REGION Network 112: SALIDAS - VELOCIDAD ANALOGICA >> RODILLOS
   // 25T229A_03 
   // Plantilla_Avance_E1S3_SinVariador_1Mesas.
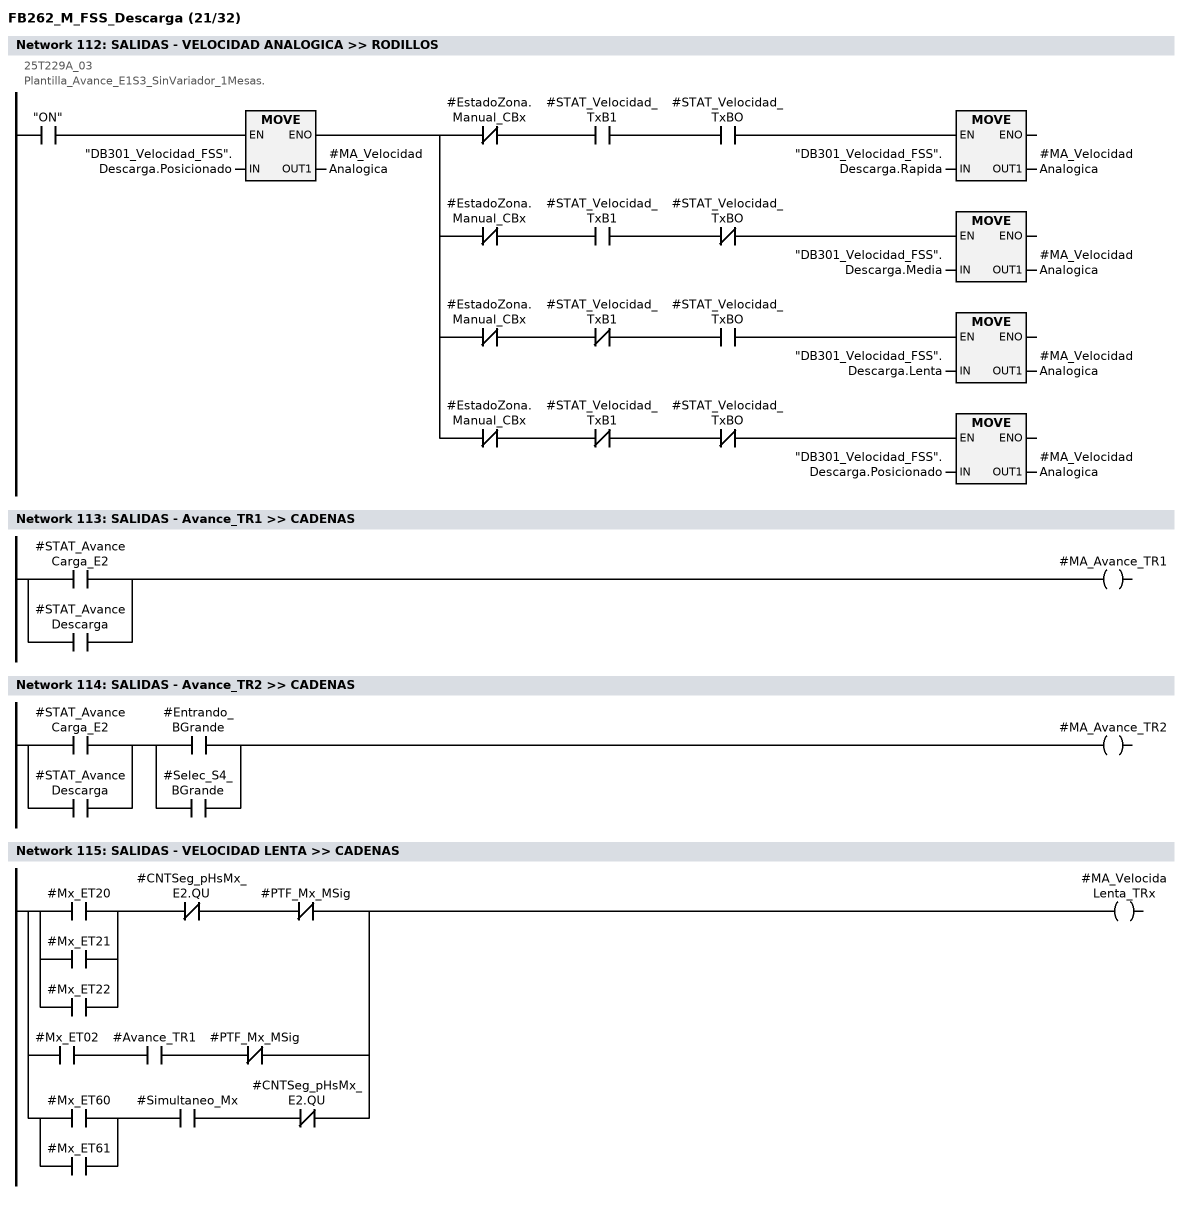
   RUNG wire#powerrail
      Contact( "ON" )
      { S7_GenerateENO := "TRUE" } Move(in := "DB301_Velocidad_FSS".Descarga.Posicionado, out1 => #MA_VelocidadAnalogica)
      wire#w1
      I_Contact( #EstadoZona.Manual_CBx )
      Contact( #STAT_Velocidad_TxB1 )
      Contact( #STAT_Velocidad_TxBO )
      { S7_GenerateENO := "TRUE" } Move(in := "DB301_Velocidad_FSS".Descarga.Rapida, out1 => #MA_VelocidadAnalogica)
   END_RUNG
   RUNG wire#w1
      I_Contact( #EstadoZona.Manual_CBx )
      Contact( #STAT_Velocidad_TxB1 )
      I_Contact( #STAT_Velocidad_TxBO )
      { S7_GenerateENO := "TRUE" } Move(in := "DB301_Velocidad_FSS".Descarga.Media, out1 => #MA_VelocidadAnalogica)
   END_RUNG
   RUNG wire#w1
      I_Contact( #EstadoZona.Manual_CBx )
      I_Contact( #STAT_Velocidad_TxB1 )
      Contact( #STAT_Velocidad_TxBO )
      { S7_GenerateENO := "TRUE" } Move(in := "DB301_Velocidad_FSS".Descarga.Lenta, out1 => #MA_VelocidadAnalogica)
   END_RUNG
   RUNG wire#w1
      I_Contact( #EstadoZona.Manual_CBx )
      I_Contact( #STAT_Velocidad_TxB1 )
      I_Contact( #STAT_Velocidad_TxBO )
      { S7_GenerateENO := "TRUE" } Move(in := "DB301_Velocidad_FSS".Descarga.Posicionado, out1 => #MA_VelocidadAnalogica)
   END_RUNG
   // the same network as SCL:
   // ENO of a box is taken as its EN; it also drops when the box reports an error
   IF "ON" THEN #MA_VelocidadAnalogica := "DB301_Velocidad_FSS".Descarga.Posicionado; END_IF;
   IF "ON" AND NOT #EstadoZona.Manual_CBx AND #STAT_Velocidad_TxB1 AND #STAT_Velocidad_TxBO THEN
       #MA_VelocidadAnalogica := "DB301_Velocidad_FSS".Descarga.Rapida;
   END_IF;
   IF "ON" AND NOT #EstadoZona.Manual_CBx AND #STAT_Velocidad_TxB1 AND NOT #STAT_Velocidad_TxBO THEN
       #MA_VelocidadAnalogica := "DB301_Velocidad_FSS".Descarga.Media;
   END_IF;
   IF "ON" AND NOT #EstadoZona.Manual_CBx AND NOT #STAT_Velocidad_TxB1 AND #STAT_Velocidad_TxBO THEN
       #MA_VelocidadAnalogica := "DB301_Velocidad_FSS".Descarga.Lenta;
   END_IF;
   IF "ON" AND NOT #EstadoZona.Manual_CBx AND NOT #STAT_Velocidad_TxB1 AND NOT #STAT_Velocidad_TxBO THEN
       #MA_VelocidadAnalogica := "DB301_Velocidad_FSS".Descarga.Posicionado;
   END_IF;
END_REGION

REGION Network 113: SALIDAS - Avance_TR1 >> CADENAS
   RUNG wire#powerrail
      Contact( #STAT_AvanceCarga_E2 )
      wire#w1
      Coil( #MA_Avance_TR1 )
   END_RUNG
   RUNG wire#powerrail
      Contact( #STAT_AvanceDescarga )
   END_RUNG wire#w1
   // the same network as SCL:
   #MA_Avance_TR1 := #STAT_AvanceCarga_E2 OR #STAT_AvanceDescarga;
END_REGION

REGION Network 114: SALIDAS - Avance_TR2 >> CADENAS
   RUNG wire#powerrail
      Contact( #STAT_AvanceCarga_E2 )
      wire#w1
      Contact( #Entrando_BGrande )
      wire#w2
      Coil( #MA_Avance_TR2 )
   END_RUNG
   RUNG wire#powerrail
      Contact( #STAT_AvanceDescarga )
   END_RUNG wire#w1
   RUNG wire#w1
      Contact( #Selec_S4_BGrande )
   END_RUNG wire#w2
   // the same network as SCL:
   #MA_Avance_TR2 := (#STAT_AvanceCarga_E2 OR #STAT_AvanceDescarga) AND (#Entrando_BGrande OR #Selec_S4_BGrande);
END_REGION

REGION Network 115: SALIDAS - VELOCIDAD LENTA >> CADENAS
   RUNG wire#powerrail
      Contact( #Mx_ET20 )
      wire#w1
      I_Contact( #CNTSeg_pHsMx_E2.QU )
      I_Contact( #PTF_Mx_MSig )
      wire#w2
      Coil( #MA_VelocidaLenta_TRx )
   END_RUNG
   RUNG wire#powerrail
      Contact( #Mx_ET21 )
   END_RUNG wire#w1
   RUNG wire#powerrail
      Contact( #Mx_ET22 )
   END_RUNG wire#w1
   RUNG wire#powerrail
      Contact( #Mx_ET02 )
      Contact( #Avance_TR1 )
      I_Contact( #PTF_Mx_MSig )
   END_RUNG wire#w2
   RUNG wire#powerrail
      Contact( #Mx_ET60 )
      wire#w3
      Contact( #Simultaneo_Mx )
      I_Contact( #CNTSeg_pHsMx_E2.QU )
   END_RUNG wire#w2
   RUNG wire#powerrail
      Contact( #Mx_ET61 )
   END_RUNG wire#w3
   // the same network as SCL:
   #MA_VelocidaLenta_TRx := ((#Mx_ET20 OR #Mx_ET21 OR #Mx_ET22) AND NOT #CNTSeg_pHsMx_E2.QU AND NOT #PTF_Mx_MSig) OR (#Mx_ET02 AND #Avance_TR1 AND NOT #PTF_Mx_MSig) OR ((#Mx_ET60 OR #Mx_ET61) AND #Simultaneo_Mx AND NOT #CNTSeg_pHsMx_E2.QU);
END_REGION

REGION Network 116: SALIDAS - SUBIR TRANSTER TR1 (Neumatica)
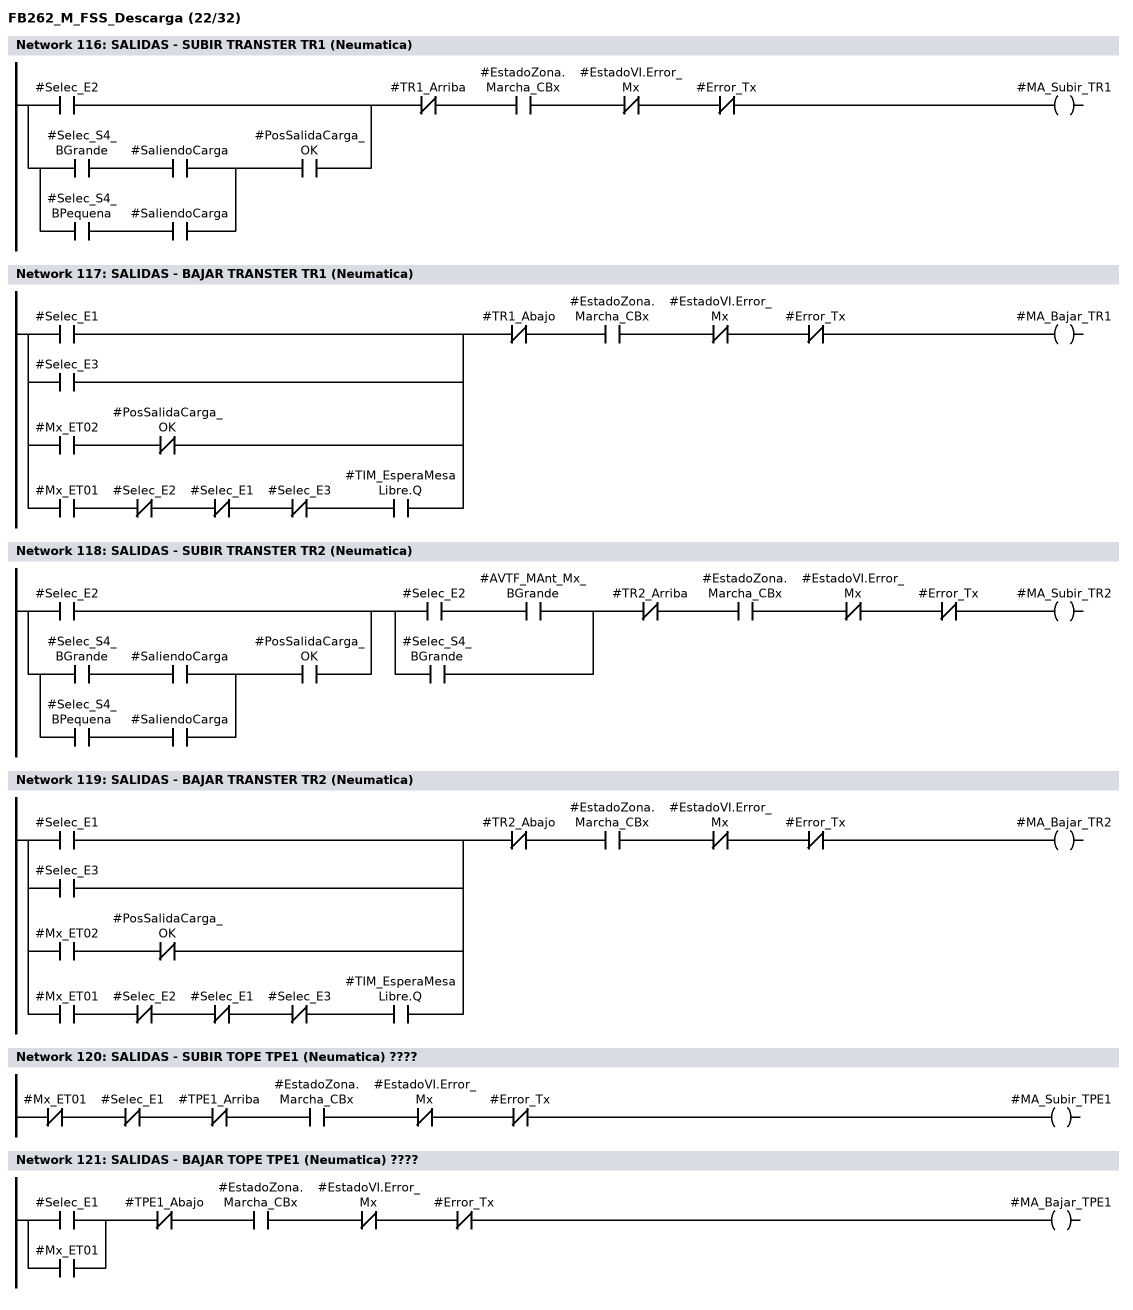
   RUNG wire#powerrail
      Contact( #Selec_E2 )
      wire#w1
      I_Contact( #TR1_Arriba )
      Contact( #EstadoZona.Marcha_CBx )
      I_Contact( #EstadoVI.Error_Mx )
      I_Contact( #Error_Tx )
      Coil( #MA_Subir_TR1 )
   END_RUNG
   RUNG wire#powerrail
      Contact( #Selec_S4_BGrande )
      Contact( #SaliendoCarga )
      wire#w2
      Contact( #PosSalidaCarga_OK )
   END_RUNG wire#w1
   RUNG wire#powerrail
      Contact( #Selec_S4_BPequena )
      Contact( #SaliendoCarga )
   END_RUNG wire#w2
   // the same network as SCL:
   #MA_Subir_TR1 := (#Selec_E2 OR (((#Selec_S4_BGrande AND #SaliendoCarga) OR (#Selec_S4_BPequena AND #SaliendoCarga)) AND #PosSalidaCarga_OK)) AND NOT #TR1_Arriba AND #EstadoZona.Marcha_CBx AND NOT #EstadoVI.Error_Mx AND NOT #Error_Tx;
END_REGION

REGION Network 117: SALIDAS - BAJAR TRANSTER TR1 (Neumatica)
   RUNG wire#powerrail
      Contact( #Selec_E1 )
      wire#w1
      I_Contact( #TR1_Abajo )
      Contact( #EstadoZona.Marcha_CBx )
      I_Contact( #EstadoVI.Error_Mx )
      I_Contact( #Error_Tx )
      Coil( #MA_Bajar_TR1 )
   END_RUNG
   RUNG wire#powerrail
      Contact( #Selec_E3 )
   END_RUNG wire#w1
   RUNG wire#powerrail
      Contact( #Mx_ET02 )
      I_Contact( #PosSalidaCarga_OK )
   END_RUNG wire#w1
   RUNG wire#powerrail
      Contact( #Mx_ET01 )
      I_Contact( #Selec_E2 )
      I_Contact( #Selec_E1 )
      I_Contact( #Selec_E3 )
      Contact( #TIM_EsperaMesaLibre.Q )
   END_RUNG wire#w1
   // the same network as SCL:
   #MA_Bajar_TR1 := (#Selec_E1 OR #Selec_E3 OR (#Mx_ET02 AND NOT #PosSalidaCarga_OK) OR (#Mx_ET01 AND NOT #Selec_E2 AND NOT #Selec_E1 AND NOT #Selec_E3 AND #TIM_EsperaMesaLibre.Q)) AND NOT #TR1_Abajo AND #EstadoZona.Marcha_CBx AND NOT #EstadoVI.Error_Mx AND NOT #Error_Tx;
END_REGION

REGION Network 118: SALIDAS - SUBIR TRANSTER TR2 (Neumatica)
   RUNG wire#powerrail
      Contact( #Selec_E2 )
      wire#w1
      Contact( #Selec_E2 )
      Contact( #AVTF_MAnt_Mx_BGrande )
      wire#w3
      I_Contact( #TR2_Arriba )
      Contact( #EstadoZona.Marcha_CBx )
      I_Contact( #EstadoVI.Error_Mx )
      I_Contact( #Error_Tx )
      Coil( #MA_Subir_TR2 )
   END_RUNG
   RUNG wire#powerrail
      Contact( #Selec_S4_BGrande )
      Contact( #SaliendoCarga )
      wire#w2
      Contact( #PosSalidaCarga_OK )
   END_RUNG wire#w1
   RUNG wire#powerrail
      Contact( #Selec_S4_BPequena )
      Contact( #SaliendoCarga )
   END_RUNG wire#w2
   RUNG wire#w1
      Contact( #Selec_S4_BGrande )
   END_RUNG wire#w3
   // the same network as SCL:
   #MA_Subir_TR2 := (#Selec_E2 OR (((#Selec_S4_BGrande AND #SaliendoCarga) OR (#Selec_S4_BPequena AND #SaliendoCarga)) AND #PosSalidaCarga_OK)) AND ((#Selec_E2 AND #AVTF_MAnt_Mx_BGrande) OR #Selec_S4_BGrande) AND NOT #TR2_Arriba AND #EstadoZona.Marcha_CBx AND NOT #EstadoVI.Error_Mx AND NOT #Error_Tx;
END_REGION

REGION Network 119: SALIDAS - BAJAR TRANSTER TR2 (Neumatica)
   RUNG wire#powerrail
      Contact( #Selec_E1 )
      wire#w1
      I_Contact( #TR2_Abajo )
      Contact( #EstadoZona.Marcha_CBx )
      I_Contact( #EstadoVI.Error_Mx )
      I_Contact( #Error_Tx )
      Coil( #MA_Bajar_TR2 )
   END_RUNG
   RUNG wire#powerrail
      Contact( #Selec_E3 )
   END_RUNG wire#w1
   RUNG wire#powerrail
      Contact( #Mx_ET02 )
      I_Contact( #PosSalidaCarga_OK )
   END_RUNG wire#w1
   RUNG wire#powerrail
      Contact( #Mx_ET01 )
      I_Contact( #Selec_E2 )
      I_Contact( #Selec_E1 )
      I_Contact( #Selec_E3 )
      Contact( #TIM_EsperaMesaLibre.Q )
   END_RUNG wire#w1
   // the same network as SCL:
   #MA_Bajar_TR2 := (#Selec_E1 OR #Selec_E3 OR (#Mx_ET02 AND NOT #PosSalidaCarga_OK) OR (#Mx_ET01 AND NOT #Selec_E2 AND NOT #Selec_E1 AND NOT #Selec_E3 AND #TIM_EsperaMesaLibre.Q)) AND NOT #TR2_Abajo AND #EstadoZona.Marcha_CBx AND NOT #EstadoVI.Error_Mx AND NOT #Error_Tx;
END_REGION

REGION Network 120: SALIDAS - SUBIR TOPE TPE1 (Neumatica) ????
   RUNG wire#powerrail
      I_Contact( #Mx_ET01 )
      I_Contact( #Selec_E1 )
      I_Contact( #TPE1_Arriba )
      Contact( #EstadoZona.Marcha_CBx )
      I_Contact( #EstadoVI.Error_Mx )
      I_Contact( #Error_Tx )
      Coil( #MA_Subir_TPE1 )
   END_RUNG
   // the same network as SCL:
   #MA_Subir_TPE1 := NOT #Mx_ET01 AND NOT #Selec_E1 AND NOT #TPE1_Arriba AND #EstadoZona.Marcha_CBx AND NOT #EstadoVI.Error_Mx AND NOT #Error_Tx;
END_REGION

REGION Network 121: SALIDAS - BAJAR TOPE TPE1 (Neumatica) ????
   RUNG wire#powerrail
      Contact( #Selec_E1 )
      wire#w1
      I_Contact( #TPE1_Abajo )
      Contact( #EstadoZona.Marcha_CBx )
      I_Contact( #EstadoVI.Error_Mx )
      I_Contact( #Error_Tx )
      Coil( #MA_Bajar_TPE1 )
   END_RUNG
   RUNG wire#powerrail
      Contact( #Mx_ET01 )
   END_RUNG wire#w1
   // the same network as SCL:
   #MA_Bajar_TPE1 := (#Selec_E1 OR #Mx_ET01) AND NOT #TPE1_Abajo AND #EstadoZona.Marcha_CBx AND NOT #EstadoVI.Error_Mx AND NOT #Error_Tx;
END_REGION

REGION Network 122: SALIDAS - SUBIR TOPE TPE3 (Neumatica) ????
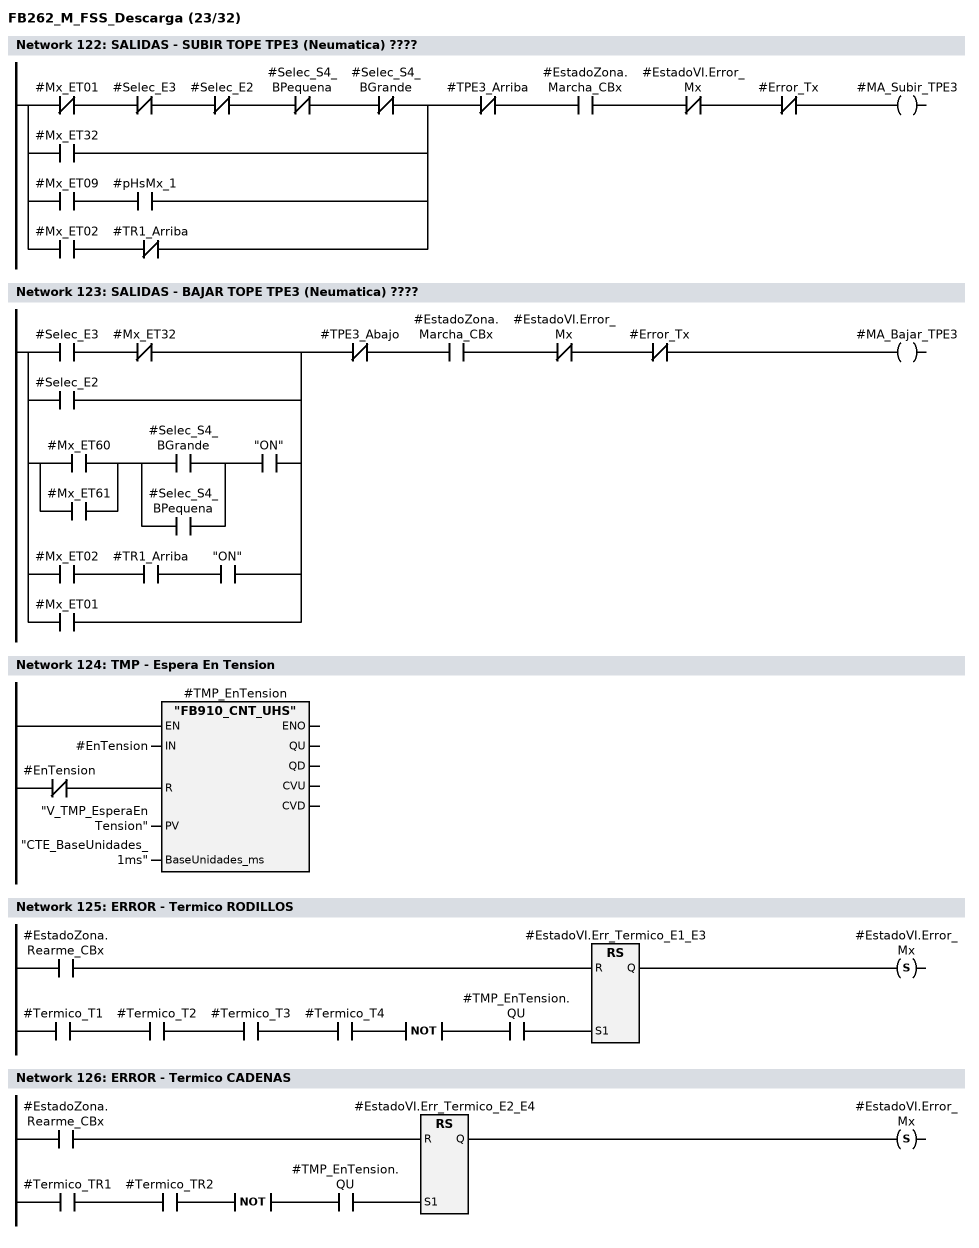
   RUNG wire#powerrail
      I_Contact( #Mx_ET01 )
      I_Contact( #Selec_E3 )
      I_Contact( #Selec_E2 )
      I_Contact( #Selec_S4_BPequena )
      I_Contact( #Selec_S4_BGrande )
      wire#w1
      I_Contact( #TPE3_Arriba )
      Contact( #EstadoZona.Marcha_CBx )
      I_Contact( #EstadoVI.Error_Mx )
      I_Contact( #Error_Tx )
      Coil( #MA_Subir_TPE3 )
   END_RUNG
   RUNG wire#powerrail
      Contact( #Mx_ET32 )
   END_RUNG wire#w1
   RUNG wire#powerrail
      Contact( #Mx_ET09 )
      Contact( #pHsMx_1 )
   END_RUNG wire#w1
   RUNG wire#powerrail
      Contact( #Mx_ET02 )
      I_Contact( #TR1_Arriba )
   END_RUNG wire#w1
   // the same network as SCL:
   #MA_Subir_TPE3 := ((NOT #Mx_ET01 AND NOT #Selec_E3 AND NOT #Selec_E2 AND NOT #Selec_S4_BPequena AND NOT #Selec_S4_BGrande) OR #Mx_ET32 OR (#Mx_ET09 AND #pHsMx_1) OR (#Mx_ET02 AND NOT #TR1_Arriba)) AND NOT #TPE3_Arriba AND #EstadoZona.Marcha_CBx AND NOT #EstadoVI.Error_Mx AND NOT #Error_Tx;
END_REGION

REGION Network 123: SALIDAS - BAJAR TOPE TPE3 (Neumatica) ????
   RUNG wire#powerrail
      Contact( #Selec_E3 )
      I_Contact( #Mx_ET32 )
      wire#w1
      I_Contact( #TPE3_Abajo )
      Contact( #EstadoZona.Marcha_CBx )
      I_Contact( #EstadoVI.Error_Mx )
      I_Contact( #Error_Tx )
      Coil( #MA_Bajar_TPE3 )
   END_RUNG
   RUNG wire#powerrail
      Contact( #Selec_E2 )
   END_RUNG wire#w1
   RUNG wire#powerrail
      Contact( #Mx_ET60 )
      wire#w2
      Contact( #Selec_S4_BGrande )
      wire#w3
      Contact( "ON" )
   END_RUNG wire#w1
   RUNG wire#powerrail
      Contact( #Mx_ET61 )
   END_RUNG wire#w2
   RUNG wire#w2
      Contact( #Selec_S4_BPequena )
   END_RUNG wire#w3
   RUNG wire#powerrail
      Contact( #Mx_ET02 )
      Contact( #TR1_Arriba )
      Contact( "ON" )
   END_RUNG wire#w1
   RUNG wire#powerrail
      Contact( #Mx_ET01 )
   END_RUNG wire#w1
   // the same network as SCL:
   #MA_Bajar_TPE3 := ((#Selec_E3 AND NOT #Mx_ET32) OR #Selec_E2 OR ((#Mx_ET60 OR #Mx_ET61) AND (#Selec_S4_BGrande OR #Selec_S4_BPequena) AND "ON") OR (#Mx_ET02 AND #TR1_Arriba AND "ON") OR #Mx_ET01) AND NOT #TPE3_Abajo AND #EstadoZona.Marcha_CBx AND NOT #EstadoVI.Error_Mx AND NOT #Error_Tx;
END_REGION

REGION Network 124: TMP - Espera En Tension
   RUNG wire#powerrail
      #TMP_EnTension(R := wire#w1, IN := #EnTension, PV := "V_TMP_EsperaEnTension", BaseUnidades_ms := "CTE_BaseUnidades_1ms", QU =>, QD =>, CVU =>, CVD =>)
   END_RUNG
   RUNG wire#powerrail
      I_Contact( #EnTension )
   END_RUNG wire#w1
   // the same network as SCL:
   #TMP_EnTension(IN := #EnTension,   // "FB910_CNT_UHS"
                  R := NOT #EnTension,
                  PV := "V_TMP_EsperaEnTension",
                  BaseUnidades_ms := "CTE_BaseUnidades_1ms");
END_REGION

REGION Network 125: ERROR - Termico RODILLOS
   RUNG wire#powerrail
      Contact( #EstadoZona.Rearme_CBx )
      S_RS(operand := #EstadoVI.Err_Termico_E1_E3, s1 := wire#w1)
      S_Coil( #EstadoVI.Error_Mx )
   END_RUNG
   RUNG wire#powerrail
      Contact( #Termico_T1 )
      Contact( #Termico_T2 )
      Contact( #Termico_T3 )
      Contact( #Termico_T4 )
      Not()
      Contact( #TMP_EnTension.QU )
   END_RUNG wire#w1
   // the same network as SCL:
   IF #EstadoZona.Rearme_CBx THEN
       #EstadoVI.Err_Termico_E1_E3 := FALSE;   // RS flip-flop
   END_IF;
   IF NOT (#Termico_T1 AND #Termico_T2 AND #Termico_T3 AND #Termico_T4) AND #TMP_EnTension.QU THEN
       #EstadoVI.Err_Termico_E1_E3 := TRUE;
   END_IF;
   IF #EstadoVI.Err_Termico_E1_E3 THEN #EstadoVI.Error_Mx := TRUE; END_IF;
END_REGION

REGION Network 126: ERROR - Termico CADENAS
   RUNG wire#powerrail
      Contact( #EstadoZona.Rearme_CBx )
      S_RS(operand := #EstadoVI.Err_Termico_E2_E4, s1 := wire#w1)
      S_Coil( #EstadoVI.Error_Mx )
   END_RUNG
   RUNG wire#powerrail
      Contact( #Termico_TR1 )
      Contact( #Termico_TR2 )
      Not()
      Contact( #TMP_EnTension.QU )
   END_RUNG wire#w1
   // the same network as SCL:
   IF #EstadoZona.Rearme_CBx THEN
       #EstadoVI.Err_Termico_E2_E4 := FALSE;   // RS flip-flop
   END_IF;
   IF NOT (#Termico_TR1 AND #Termico_TR2) AND #TMP_EnTension.QU THEN
       #EstadoVI.Err_Termico_E2_E4 := TRUE;
   END_IF;
   IF #EstadoVI.Err_Termico_E2_E4 THEN #EstadoVI.Error_Mx := TRUE; END_IF;
END_REGION

REGION Network 127: ERROR - Mesa Ocupada
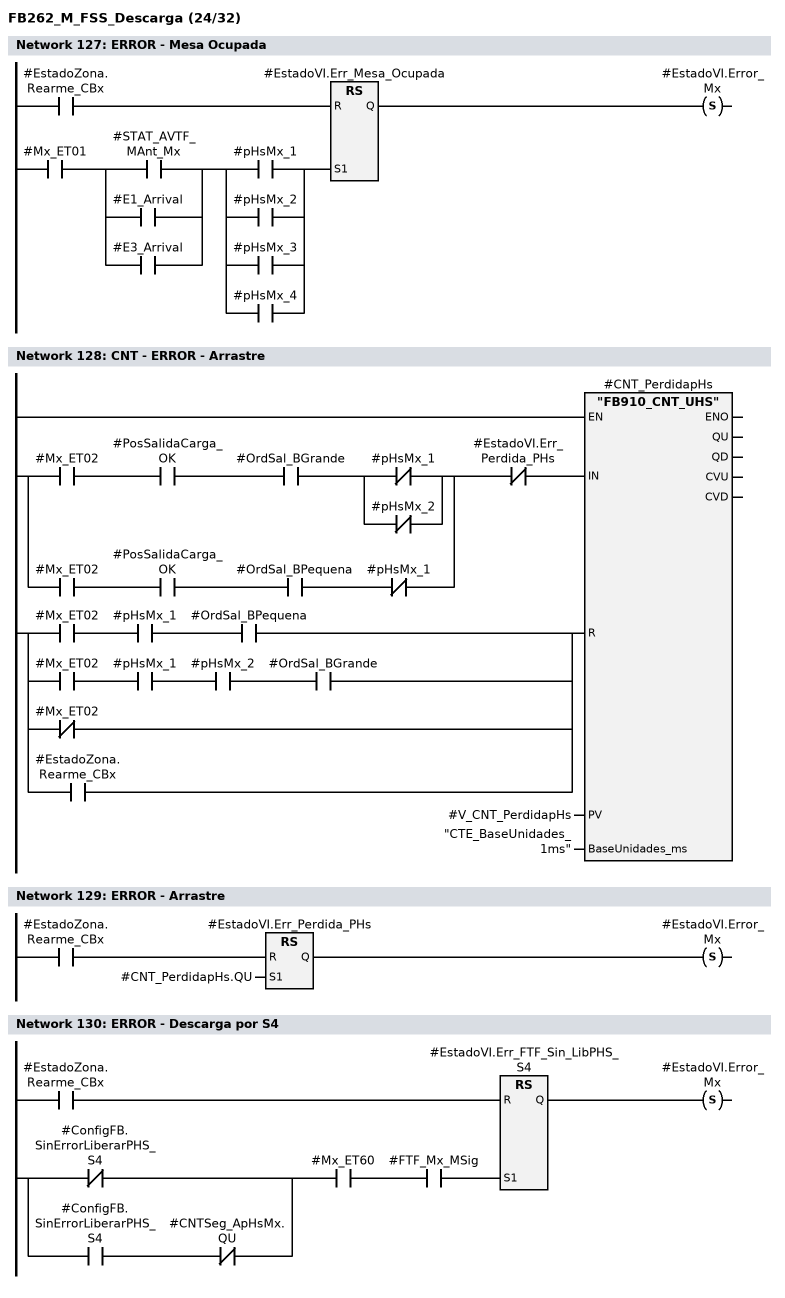
   RUNG wire#powerrail
      Contact( #EstadoZona.Rearme_CBx )
      S_RS(operand := #EstadoVI.Err_Mesa_Ocupada, s1 := wire#w3)
      S_Coil( #EstadoVI.Error_Mx )
   END_RUNG
   RUNG wire#powerrail
      Contact( #Mx_ET01 )
      wire#w1
      Contact( #STAT_AVTF_MAnt_Mx )
      wire#w2
      Contact( #pHsMx_1 )
   END_RUNG wire#w3
   RUNG wire#w1
      Contact( #E1_Arrival )
   END_RUNG wire#w2
   RUNG wire#w1
      Contact( #E3_Arrival )
   END_RUNG wire#w2
   RUNG wire#w2
      Contact( #pHsMx_2 )
   END_RUNG wire#w3
   RUNG wire#w2
      Contact( #pHsMx_3 )
   END_RUNG wire#w3
   RUNG wire#w2
      Contact( #pHsMx_4 )
   END_RUNG wire#w3
   // the same network as SCL:
   IF #EstadoZona.Rearme_CBx THEN
       #EstadoVI.Err_Mesa_Ocupada := FALSE;   // RS flip-flop
   END_IF;
   IF #Mx_ET01 AND (#STAT_AVTF_MAnt_Mx OR #E1_Arrival OR #E3_Arrival) AND (#pHsMx_1 OR #pHsMx_2 OR #pHsMx_3 OR #pHsMx_4) THEN
       #EstadoVI.Err_Mesa_Ocupada := TRUE;
   END_IF;
   IF #EstadoVI.Err_Mesa_Ocupada THEN #EstadoVI.Error_Mx := TRUE; END_IF;
END_REGION

REGION Network 128: CNT - ERROR - Arrastre
   RUNG wire#powerrail
      #CNT_PerdidapHs(IN := wire#w3, R := wire#w4, PV := #V_CNT_PerdidapHs, BaseUnidades_ms := "CTE_BaseUnidades_1ms", QU =>, QD =>, CVU =>, CVD =>)
   END_RUNG
   RUNG wire#powerrail
      Contact( #Mx_ET02 )
      Contact( #PosSalidaCarga_OK )
      Contact( #OrdSal_BGrande )
      wire#w1
      I_Contact( #pHsMx_1 )
      wire#w2
      I_Contact( #EstadoVI.Err_Perdida_PHs )
   END_RUNG wire#w3
   RUNG wire#w1
      I_Contact( #pHsMx_2 )
   END_RUNG wire#w2
   RUNG wire#powerrail
      Contact( #Mx_ET02 )
      Contact( #PosSalidaCarga_OK )
      Contact( #OrdSal_BPequena )
      I_Contact( #pHsMx_1 )
   END_RUNG wire#w2
   RUNG wire#powerrail
      Contact( #Mx_ET02 )
      Contact( #pHsMx_1 )
      Contact( #OrdSal_BPequena )
   END_RUNG wire#w4
   RUNG wire#powerrail
      Contact( #Mx_ET02 )
      Contact( #pHsMx_1 )
      Contact( #pHsMx_2 )
      Contact( #OrdSal_BGrande )
   END_RUNG wire#w4
   RUNG wire#powerrail
      I_Contact( #Mx_ET02 )
   END_RUNG wire#w4
   RUNG wire#powerrail
      Contact( #EstadoZona.Rearme_CBx )
   END_RUNG wire#w4
   // the same network as SCL:
   #CNT_PerdidapHs(IN := ((#Mx_ET02 AND #PosSalidaCarga_OK AND #OrdSal_BGrande AND (NOT #pHsMx_1 OR NOT #pHsMx_2)) OR (#Mx_ET02 AND #PosSalidaCarga_OK AND #OrdSal_BPequena AND NOT #pHsMx_1)) AND NOT #EstadoVI.Err_Perdida_PHs,   // "FB910_CNT_UHS"
                   R := (#Mx_ET02 AND #pHsMx_1 AND #OrdSal_BPequena) OR (#Mx_ET02 AND #pHsMx_1 AND #pHsMx_2 AND #OrdSal_BGrande) OR NOT #Mx_ET02 OR #EstadoZona.Rearme_CBx,
                   PV := #V_CNT_PerdidapHs,
                   BaseUnidades_ms := "CTE_BaseUnidades_1ms");
END_REGION

REGION Network 129: ERROR - Arrastre
   RUNG wire#powerrail
      Contact( #EstadoZona.Rearme_CBx )
      S_RS(operand := #EstadoVI.Err_Perdida_PHs, s1 := #CNT_PerdidapHs.QU)
      S_Coil( #EstadoVI.Error_Mx )
   END_RUNG
   // the same network as SCL:
   IF #EstadoZona.Rearme_CBx THEN
       #EstadoVI.Err_Perdida_PHs := FALSE;   // RS flip-flop
   END_IF;
   IF #CNT_PerdidapHs.QU THEN #EstadoVI.Err_Perdida_PHs := TRUE; END_IF;
   IF #EstadoVI.Err_Perdida_PHs THEN #EstadoVI.Error_Mx := TRUE; END_IF;
END_REGION

REGION Network 130: ERROR - Descarga por S4
   RUNG wire#powerrail
      Contact( #EstadoZona.Rearme_CBx )
      S_RS(operand := #EstadoVI.Err_FTF_Sin_LibPHS_S4, s1 := wire#w2)
      S_Coil( #EstadoVI.Error_Mx )
   END_RUNG
   RUNG wire#powerrail
      I_Contact( #ConfigFB.SinErrorLiberarPHS_S4 )
      wire#w1
      Contact( #Mx_ET60 )
      Contact( #FTF_Mx_MSig )
   END_RUNG wire#w2
   RUNG wire#powerrail
      Contact( #ConfigFB.SinErrorLiberarPHS_S4 )
      I_Contact( #CNTSeg_ApHsMx.QU )
   END_RUNG wire#w1
   // the same network as SCL:
   IF #EstadoZona.Rearme_CBx THEN
       #EstadoVI.Err_FTF_Sin_LibPHS_S4 := FALSE;   // RS flip-flop
   END_IF;
   IF (NOT #ConfigFB.SinErrorLiberarPHS_S4 OR (#ConfigFB.SinErrorLiberarPHS_S4 AND NOT #CNTSeg_ApHsMx.QU)) AND #Mx_ET60 AND #FTF_Mx_MSig THEN
       #EstadoVI.Err_FTF_Sin_LibPHS_S4 := TRUE;
   END_IF;
   IF #EstadoVI.Err_FTF_Sin_LibPHS_S4 THEN #EstadoVI.Error_Mx := TRUE; END_IF;
END_REGION

REGION Network 131: TMP - ERROR - TimeOut Avance Tx >>> DESCARGA FSS Y REPOSICONADO
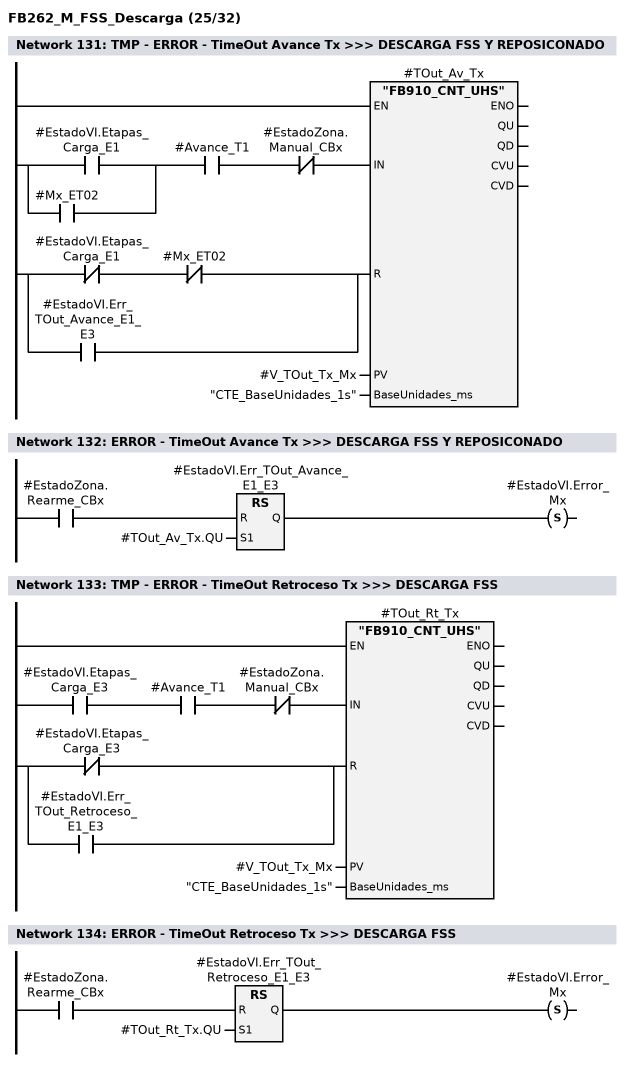
   RUNG wire#powerrail
      #TOut_Av_Tx(IN := wire#w2, R := wire#w3, PV := #V_TOut_Tx_Mx, BaseUnidades_ms := "CTE_BaseUnidades_1s", QU =>, QD =>, CVU =>, CVD =>)
   END_RUNG
   RUNG wire#powerrail
      Contact( #EstadoVI.Etapas_Carga_E1 )
      wire#w1
      Contact( #Avance_T1 )
      I_Contact( #EstadoZona.Manual_CBx )
   END_RUNG wire#w2
   RUNG wire#powerrail
      Contact( #Mx_ET02 )
   END_RUNG wire#w1
   RUNG wire#powerrail
      I_Contact( #EstadoVI.Etapas_Carga_E1 )
      I_Contact( #Mx_ET02 )
   END_RUNG wire#w3
   RUNG wire#powerrail
      Contact( #EstadoVI.Err_TOut_Avance_E1_E3 )
   END_RUNG wire#w3
   // the same network as SCL:
   #TOut_Av_Tx(IN := (#EstadoVI.Etapas_Carga_E1 OR #Mx_ET02) AND #Avance_T1 AND NOT #EstadoZona.Manual_CBx,   // "FB910_CNT_UHS"
               R := (NOT #EstadoVI.Etapas_Carga_E1 AND NOT #Mx_ET02) OR #EstadoVI.Err_TOut_Avance_E1_E3,
               PV := #V_TOut_Tx_Mx,
               BaseUnidades_ms := "CTE_BaseUnidades_1s");
END_REGION

REGION Network 132: ERROR - TimeOut Avance Tx >>> DESCARGA FSS Y REPOSICONADO
   RUNG wire#powerrail
      Contact( #EstadoZona.Rearme_CBx )
      S_RS(operand := #EstadoVI.Err_TOut_Avance_E1_E3, s1 := #TOut_Av_Tx.QU)
      S_Coil( #EstadoVI.Error_Mx )
   END_RUNG
   // the same network as SCL:
   IF #EstadoZona.Rearme_CBx THEN
       #EstadoVI.Err_TOut_Avance_E1_E3 := FALSE;   // RS flip-flop
   END_IF;
   IF #TOut_Av_Tx.QU THEN #EstadoVI.Err_TOut_Avance_E1_E3 := TRUE; END_IF;
   IF #EstadoVI.Err_TOut_Avance_E1_E3 THEN #EstadoVI.Error_Mx := TRUE; END_IF;
END_REGION

REGION Network 133: TMP - ERROR - TimeOut Retroceso Tx >>> DESCARGA FSS
   RUNG wire#powerrail
      #TOut_Rt_Tx(IN := wire#w1, R := wire#w2, PV := #V_TOut_Tx_Mx, BaseUnidades_ms := "CTE_BaseUnidades_1s", QU =>, QD =>, CVU =>, CVD =>)
   END_RUNG
   RUNG wire#powerrail
      Contact( #EstadoVI.Etapas_Carga_E3 )
      Contact( #Avance_T1 )
      I_Contact( #EstadoZona.Manual_CBx )
   END_RUNG wire#w1
   RUNG wire#powerrail
      I_Contact( #EstadoVI.Etapas_Carga_E3 )
   END_RUNG wire#w2
   RUNG wire#powerrail
      Contact( #EstadoVI.Err_TOut_Retroceso_E1_E3 )
   END_RUNG wire#w2
   // the same network as SCL:
   #TOut_Rt_Tx(IN := #EstadoVI.Etapas_Carga_E3 AND #Avance_T1 AND NOT #EstadoZona.Manual_CBx,   // "FB910_CNT_UHS"
               R := NOT #EstadoVI.Etapas_Carga_E3 OR #EstadoVI.Err_TOut_Retroceso_E1_E3,
               PV := #V_TOut_Tx_Mx,
               BaseUnidades_ms := "CTE_BaseUnidades_1s");
END_REGION

REGION Network 134: ERROR - TimeOut Retroceso Tx >>> DESCARGA FSS
   RUNG wire#powerrail
      Contact( #EstadoZona.Rearme_CBx )
      S_RS(operand := #EstadoVI.Err_TOut_Retroceso_E1_E3, s1 := #TOut_Rt_Tx.QU)
      S_Coil( #EstadoVI.Error_Mx )
   END_RUNG
   // the same network as SCL:
   IF #EstadoZona.Rearme_CBx THEN
       #EstadoVI.Err_TOut_Retroceso_E1_E3 := FALSE;   // RS flip-flop
   END_IF;
   IF #TOut_Rt_Tx.QU THEN #EstadoVI.Err_TOut_Retroceso_E1_E3 := TRUE; END_IF;
   IF #EstadoVI.Err_TOut_Retroceso_E1_E3 THEN #EstadoVI.Error_Mx := TRUE; END_IF;
END_REGION

REGION Network 135: TMP - ERROR - TimeOut Avance TRx >>> ENTRADA
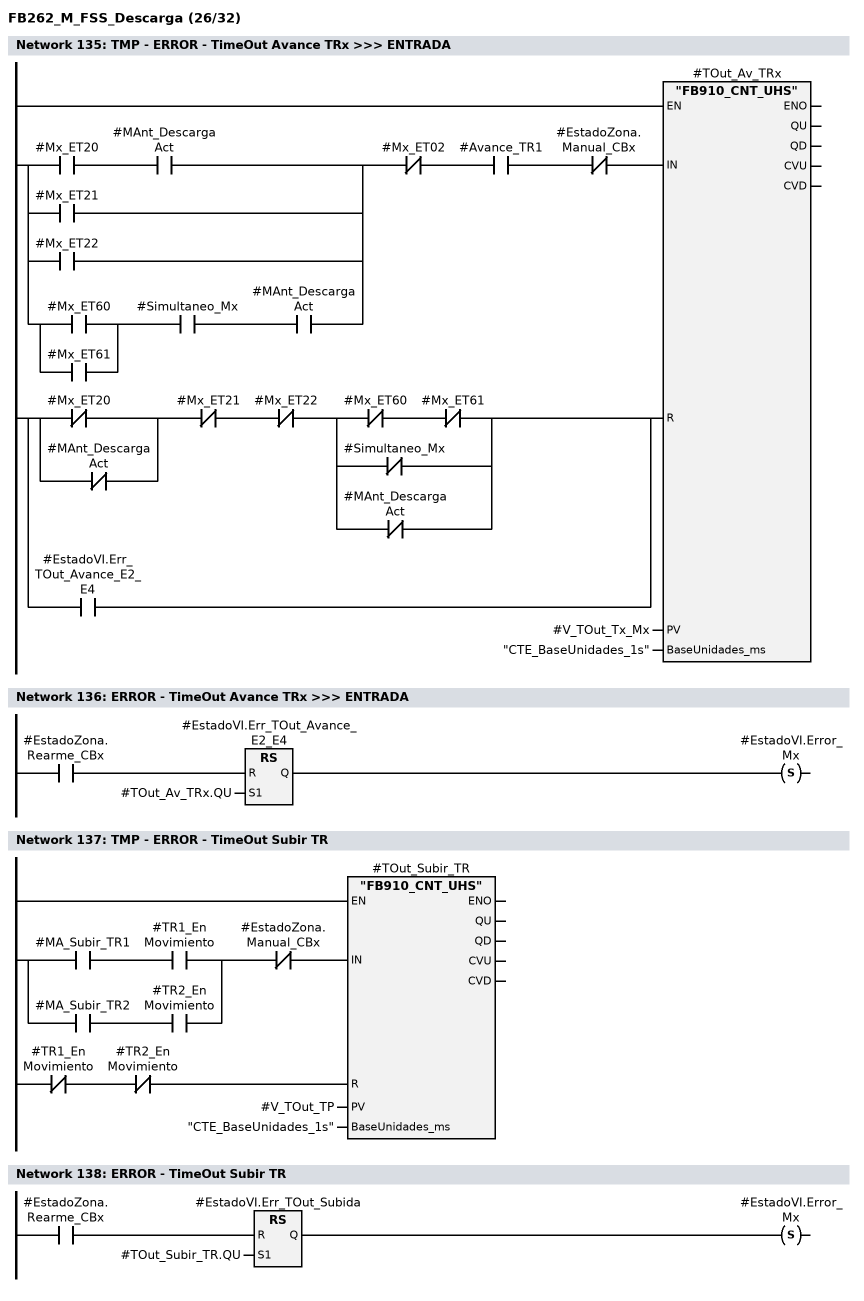
   RUNG wire#powerrail
      #TOut_Av_TRx(IN := wire#w3, R := wire#w6, PV := #V_TOut_Tx_Mx, BaseUnidades_ms := "CTE_BaseUnidades_1s", QU =>, QD =>, CVU =>, CVD =>)
   END_RUNG
   RUNG wire#powerrail
      Contact( #Mx_ET20 )
      Contact( #MAnt_DescargaAct )
      wire#w1
      I_Contact( #Mx_ET02 )
      Contact( #Avance_TR1 )
      I_Contact( #EstadoZona.Manual_CBx )
   END_RUNG wire#w3
   RUNG wire#powerrail
      Contact( #Mx_ET21 )
   END_RUNG wire#w1
   RUNG wire#powerrail
      Contact( #Mx_ET22 )
   END_RUNG wire#w1
   RUNG wire#powerrail
      Contact( #Mx_ET60 )
      wire#w2
      Contact( #Simultaneo_Mx )
      Contact( #MAnt_DescargaAct )
   END_RUNG wire#w1
   RUNG wire#powerrail
      Contact( #Mx_ET61 )
   END_RUNG wire#w2
   RUNG wire#powerrail
      I_Contact( #Mx_ET20 )
      wire#w4
      I_Contact( #Mx_ET21 )
      I_Contact( #Mx_ET22 )
      wire#w5
      I_Contact( #Mx_ET60 )
      I_Contact( #Mx_ET61 )
   END_RUNG wire#w6
   RUNG wire#powerrail
      I_Contact( #MAnt_DescargaAct )
   END_RUNG wire#w4
   RUNG wire#w5
      I_Contact( #Simultaneo_Mx )
   END_RUNG wire#w6
   RUNG wire#w5
      I_Contact( #MAnt_DescargaAct )
   END_RUNG wire#w6
   RUNG wire#powerrail
      Contact( #EstadoVI.Err_TOut_Avance_E2_E4 )
   END_RUNG wire#w6
   // the same network as SCL:
   #TOut_Av_TRx(IN := ((#Mx_ET20 AND #MAnt_DescargaAct) OR #Mx_ET21 OR #Mx_ET22 OR ((#Mx_ET60 OR #Mx_ET61) AND #Simultaneo_Mx AND #MAnt_DescargaAct)) AND NOT #Mx_ET02 AND #Avance_TR1 AND NOT #EstadoZona.Manual_CBx,   // "FB910_CNT_UHS"
                R := ((NOT #Mx_ET20 OR NOT #MAnt_DescargaAct) AND NOT #Mx_ET21 AND NOT #Mx_ET22 AND ((NOT #Mx_ET60 AND NOT #Mx_ET61) OR NOT #Simultaneo_Mx OR NOT #MAnt_DescargaAct)) OR #EstadoVI.Err_TOut_Avance_E2_E4,
                PV := #V_TOut_Tx_Mx,
                BaseUnidades_ms := "CTE_BaseUnidades_1s");
END_REGION

REGION Network 136: ERROR - TimeOut Avance TRx >>> ENTRADA
   RUNG wire#powerrail
      Contact( #EstadoZona.Rearme_CBx )
      S_RS(operand := #EstadoVI.Err_TOut_Avance_E2_E4, s1 := #TOut_Av_TRx.QU)
      S_Coil( #EstadoVI.Error_Mx )
   END_RUNG
   // the same network as SCL:
   IF #EstadoZona.Rearme_CBx THEN
       #EstadoVI.Err_TOut_Avance_E2_E4 := FALSE;   // RS flip-flop
   END_IF;
   IF #TOut_Av_TRx.QU THEN #EstadoVI.Err_TOut_Avance_E2_E4 := TRUE; END_IF;
   IF #EstadoVI.Err_TOut_Avance_E2_E4 THEN #EstadoVI.Error_Mx := TRUE; END_IF;
END_REGION

REGION Network 137: TMP - ERROR - TimeOut Subir TR
   RUNG wire#powerrail
      #TOut_Subir_TR(IN := wire#w2, R := wire#w3, PV := #V_TOut_TP, BaseUnidades_ms := "CTE_BaseUnidades_1s", QU =>, QD =>, CVU =>, CVD =>)
   END_RUNG
   RUNG wire#powerrail
      Contact( #MA_Subir_TR1 )
      Contact( #TR1_EnMovimiento )
      wire#w1
      I_Contact( #EstadoZona.Manual_CBx )
   END_RUNG wire#w2
   RUNG wire#powerrail
      Contact( #MA_Subir_TR2 )
      Contact( #TR2_EnMovimiento )
   END_RUNG wire#w1
   RUNG wire#powerrail
      I_Contact( #TR1_EnMovimiento )
      I_Contact( #TR2_EnMovimiento )
   END_RUNG wire#w3
   // the same network as SCL:
   #TOut_Subir_TR(IN := ((#MA_Subir_TR1 AND #TR1_EnMovimiento) OR (#MA_Subir_TR2 AND #TR2_EnMovimiento)) AND NOT #EstadoZona.Manual_CBx,   // "FB910_CNT_UHS"
                  R := NOT #TR1_EnMovimiento AND NOT #TR2_EnMovimiento,
                  PV := #V_TOut_TP,
                  BaseUnidades_ms := "CTE_BaseUnidades_1s");
END_REGION

REGION Network 138: ERROR - TimeOut Subir TR
   RUNG wire#powerrail
      Contact( #EstadoZona.Rearme_CBx )
      S_RS(operand := #EstadoVI.Err_TOut_Subida, s1 := #TOut_Subir_TR.QU)
      S_Coil( #EstadoVI.Error_Mx )
   END_RUNG
   // the same network as SCL:
   IF #EstadoZona.Rearme_CBx THEN
       #EstadoVI.Err_TOut_Subida := FALSE;   // RS flip-flop
   END_IF;
   IF #TOut_Subir_TR.QU THEN #EstadoVI.Err_TOut_Subida := TRUE; END_IF;
   IF #EstadoVI.Err_TOut_Subida THEN #EstadoVI.Error_Mx := TRUE; END_IF;
END_REGION

REGION Network 139: TMP - ERROR - TimeOut Bajar TR
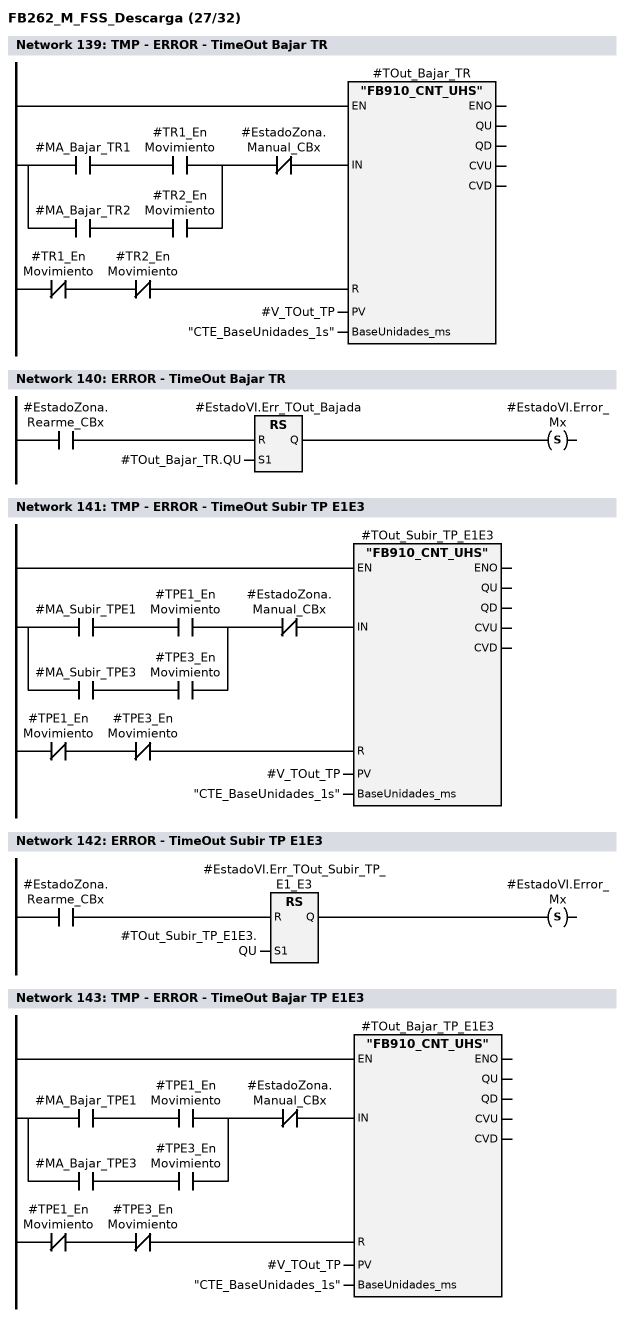
   RUNG wire#powerrail
      #TOut_Bajar_TR(IN := wire#w2, R := wire#w3, PV := #V_TOut_TP, BaseUnidades_ms := "CTE_BaseUnidades_1s", QU =>, QD =>, CVU =>, CVD =>)
   END_RUNG
   RUNG wire#powerrail
      Contact( #MA_Bajar_TR1 )
      Contact( #TR1_EnMovimiento )
      wire#w1
      I_Contact( #EstadoZona.Manual_CBx )
   END_RUNG wire#w2
   RUNG wire#powerrail
      Contact( #MA_Bajar_TR2 )
      Contact( #TR2_EnMovimiento )
   END_RUNG wire#w1
   RUNG wire#powerrail
      I_Contact( #TR1_EnMovimiento )
      I_Contact( #TR2_EnMovimiento )
   END_RUNG wire#w3
   // the same network as SCL:
   #TOut_Bajar_TR(IN := ((#MA_Bajar_TR1 AND #TR1_EnMovimiento) OR (#MA_Bajar_TR2 AND #TR2_EnMovimiento)) AND NOT #EstadoZona.Manual_CBx,   // "FB910_CNT_UHS"
                  R := NOT #TR1_EnMovimiento AND NOT #TR2_EnMovimiento,
                  PV := #V_TOut_TP,
                  BaseUnidades_ms := "CTE_BaseUnidades_1s");
END_REGION

REGION Network 140: ERROR - TimeOut Bajar TR
   RUNG wire#powerrail
      Contact( #EstadoZona.Rearme_CBx )
      S_RS(operand := #EstadoVI.Err_TOut_Bajada, s1 := #TOut_Bajar_TR.QU)
      S_Coil( #EstadoVI.Error_Mx )
   END_RUNG
   // the same network as SCL:
   IF #EstadoZona.Rearme_CBx THEN
       #EstadoVI.Err_TOut_Bajada := FALSE;   // RS flip-flop
   END_IF;
   IF #TOut_Bajar_TR.QU THEN #EstadoVI.Err_TOut_Bajada := TRUE; END_IF;
   IF #EstadoVI.Err_TOut_Bajada THEN #EstadoVI.Error_Mx := TRUE; END_IF;
END_REGION

REGION Network 141: TMP - ERROR - TimeOut Subir TP E1E3
   RUNG wire#powerrail
      #TOut_Subir_TP_E1E3(IN := wire#w2, R := wire#w3, PV := #V_TOut_TP, BaseUnidades_ms := "CTE_BaseUnidades_1s", QU =>, QD =>, CVU =>, CVD =>)
   END_RUNG
   RUNG wire#powerrail
      Contact( #MA_Subir_TPE1 )
      Contact( #TPE1_EnMovimiento )
      wire#w1
      I_Contact( #EstadoZona.Manual_CBx )
   END_RUNG wire#w2
   RUNG wire#powerrail
      Contact( #MA_Subir_TPE3 )
      Contact( #TPE3_EnMovimiento )
   END_RUNG wire#w1
   RUNG wire#powerrail
      I_Contact( #TPE1_EnMovimiento )
      I_Contact( #TPE3_EnMovimiento )
   END_RUNG wire#w3
   // the same network as SCL:
   #TOut_Subir_TP_E1E3(IN := ((#MA_Subir_TPE1 AND #TPE1_EnMovimiento) OR (#MA_Subir_TPE3 AND #TPE3_EnMovimiento)) AND NOT #EstadoZona.Manual_CBx,   // "FB910_CNT_UHS"
                       R := NOT #TPE1_EnMovimiento AND NOT #TPE3_EnMovimiento,
                       PV := #V_TOut_TP,
                       BaseUnidades_ms := "CTE_BaseUnidades_1s");
END_REGION

REGION Network 142: ERROR - TimeOut Subir TP E1E3
   RUNG wire#powerrail
      Contact( #EstadoZona.Rearme_CBx )
      S_RS(operand := #EstadoVI.Err_TOut_Subir_TP_E1_E3, s1 := #TOut_Subir_TP_E1E3.QU)
      S_Coil( #EstadoVI.Error_Mx )
   END_RUNG
   // the same network as SCL:
   IF #EstadoZona.Rearme_CBx THEN
       #EstadoVI.Err_TOut_Subir_TP_E1_E3 := FALSE;   // RS flip-flop
   END_IF;
   IF #TOut_Subir_TP_E1E3.QU THEN #EstadoVI.Err_TOut_Subir_TP_E1_E3 := TRUE; END_IF;
   IF #EstadoVI.Err_TOut_Subir_TP_E1_E3 THEN #EstadoVI.Error_Mx := TRUE; END_IF;
END_REGION

REGION Network 143: TMP - ERROR - TimeOut Bajar TP E1E3
   RUNG wire#powerrail
      #TOut_Bajar_TP_E1E3(IN := wire#w2, R := wire#w3, PV := #V_TOut_TP, BaseUnidades_ms := "CTE_BaseUnidades_1s", QU =>, QD =>, CVU =>, CVD =>)
   END_RUNG
   RUNG wire#powerrail
      Contact( #MA_Bajar_TPE1 )
      Contact( #TPE1_EnMovimiento )
      wire#w1
      I_Contact( #EstadoZona.Manual_CBx )
   END_RUNG wire#w2
   RUNG wire#powerrail
      Contact( #MA_Bajar_TPE3 )
      Contact( #TPE3_EnMovimiento )
   END_RUNG wire#w1
   RUNG wire#powerrail
      I_Contact( #TPE1_EnMovimiento )
      I_Contact( #TPE3_EnMovimiento )
   END_RUNG wire#w3
   // the same network as SCL:
   #TOut_Bajar_TP_E1E3(IN := ((#MA_Bajar_TPE1 AND #TPE1_EnMovimiento) OR (#MA_Bajar_TPE3 AND #TPE3_EnMovimiento)) AND NOT #EstadoZona.Manual_CBx,   // "FB910_CNT_UHS"
                       R := NOT #TPE1_EnMovimiento AND NOT #TPE3_EnMovimiento,
                       PV := #V_TOut_TP,
                       BaseUnidades_ms := "CTE_BaseUnidades_1s");
END_REGION

REGION Network 144: ERROR - TimeOut Bajar TP E1E3
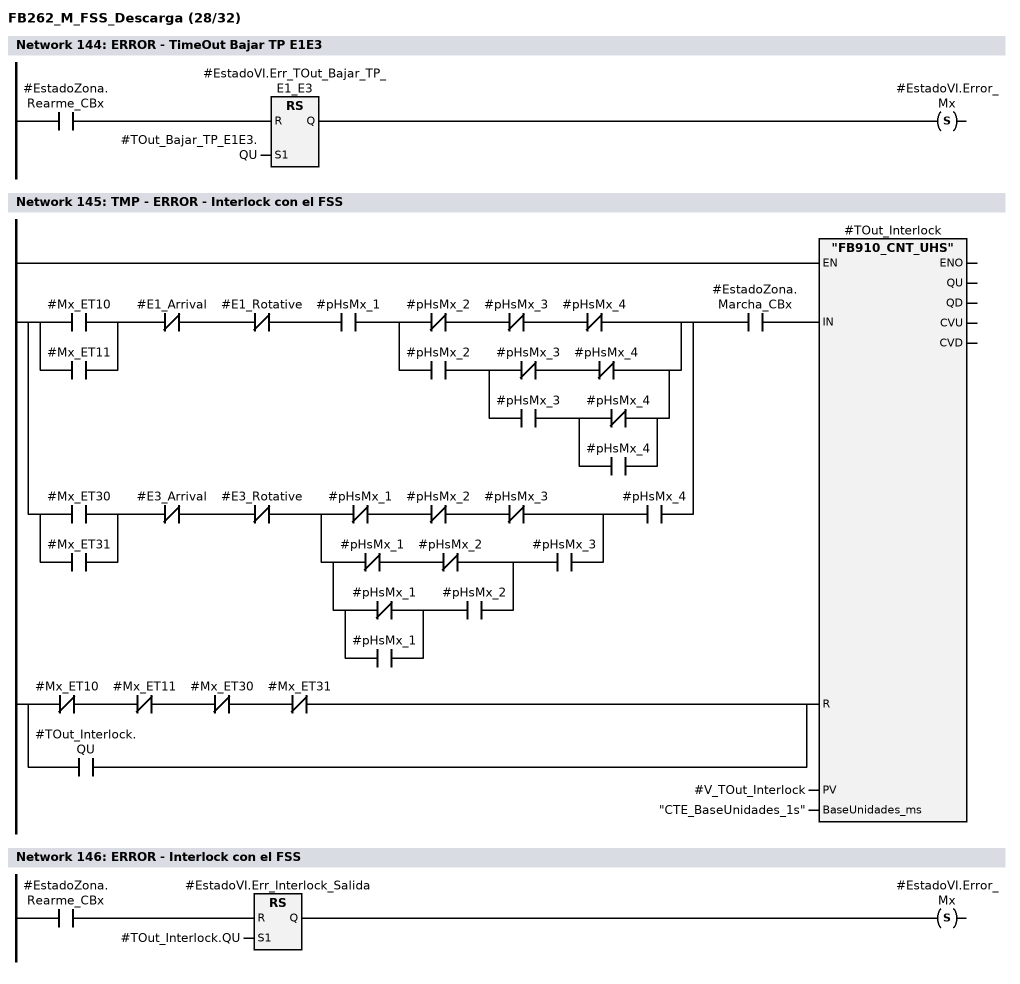
   RUNG wire#powerrail
      Contact( #EstadoZona.Rearme_CBx )
      S_RS(operand := #EstadoVI.Err_TOut_Bajar_TP_E1_E3, s1 := #TOut_Bajar_TP_E1E3.QU)
      S_Coil( #EstadoVI.Error_Mx )
   END_RUNG
   // the same network as SCL:
   IF #EstadoZona.Rearme_CBx THEN
       #EstadoVI.Err_TOut_Bajar_TP_E1_E3 := FALSE;   // RS flip-flop
   END_IF;
   IF #TOut_Bajar_TP_E1E3.QU THEN #EstadoVI.Err_TOut_Bajar_TP_E1_E3 := TRUE; END_IF;
   IF #EstadoVI.Err_TOut_Bajar_TP_E1_E3 THEN #EstadoVI.Error_Mx := TRUE; END_IF;
END_REGION

REGION Network 145: TMP - ERROR - Interlock con el FSS
   RUNG wire#powerrail
      #TOut_Interlock(IN := wire#w11, R := wire#w12, PV := #V_TOut_Interlock, BaseUnidades_ms := "CTE_BaseUnidades_1s", QU =>, QD =>, CVU =>, CVD =>)
   END_RUNG
   RUNG wire#powerrail
      Contact( #Mx_ET10 )
      wire#w1
      I_Contact( #E1_Arrival )
      I_Contact( #E1_Rotative )
      Contact( #pHsMx_1 )
      wire#w2
      I_Contact( #pHsMx_2 )
      I_Contact( #pHsMx_3 )
      I_Contact( #pHsMx_4 )
      wire#w3
      Contact( #EstadoZona.Marcha_CBx )
   END_RUNG wire#w11
   RUNG wire#powerrail
      Contact( #Mx_ET11 )
   END_RUNG wire#w1
   RUNG wire#w2
      Contact( #pHsMx_2 )
      wire#w4
      I_Contact( #pHsMx_3 )
      I_Contact( #pHsMx_4 )
   END_RUNG wire#w3
   RUNG wire#w4
      Contact( #pHsMx_3 )
      wire#w5
      I_Contact( #pHsMx_4 )
   END_RUNG wire#w3
   RUNG wire#w5
      Contact( #pHsMx_4 )
   END_RUNG wire#w3
   RUNG wire#powerrail
      Contact( #Mx_ET30 )
      wire#w6
      I_Contact( #E3_Arrival )
      I_Contact( #E3_Rotative )
      wire#w7
      I_Contact( #pHsMx_1 )
      I_Contact( #pHsMx_2 )
      I_Contact( #pHsMx_3 )
      wire#w8
      Contact( #pHsMx_4 )
   END_RUNG wire#w3
   RUNG wire#powerrail
      Contact( #Mx_ET31 )
   END_RUNG wire#w6
   RUNG wire#w7
      I_Contact( #pHsMx_1 )
      I_Contact( #pHsMx_2 )
      wire#w9
      Contact( #pHsMx_3 )
   END_RUNG wire#w8
   RUNG wire#w7
      I_Contact( #pHsMx_1 )
      wire#w10
      Contact( #pHsMx_2 )
   END_RUNG wire#w9
   RUNG wire#w7
      Contact( #pHsMx_1 )
   END_RUNG wire#w10
   RUNG wire#powerrail
      I_Contact( #Mx_ET10 )
      I_Contact( #Mx_ET11 )
      I_Contact( #Mx_ET30 )
      I_Contact( #Mx_ET31 )
   END_RUNG wire#w12
   RUNG wire#powerrail
      Contact( #TOut_Interlock.QU )
   END_RUNG wire#w12
   // the same network as SCL:
   #TOut_Interlock(IN := (((#Mx_ET10 OR #Mx_ET11) AND NOT #E1_Arrival AND NOT #E1_Rotative AND #pHsMx_1 AND ((NOT #pHsMx_2 AND NOT #pHsMx_3 AND NOT #pHsMx_4) OR (#pHsMx_2 AND ((NOT #pHsMx_3 AND NOT #pHsMx_4) OR (#pHsMx_3 AND (NOT #pHsMx_4 OR #pHsMx_4)))))) OR ((#Mx_ET30 OR #Mx_ET31) AND NOT #E3_Arrival AND NOT #E3_Rotative AND ((NOT #pHsMx_1 AND NOT #pHsMx_2 AND NOT #pHsMx_3) OR (((NOT #pHsMx_1 AND NOT #pHsMx_2) OR ((NOT #pHsMx_1 OR #pHsMx_1) AND #pHsMx_2)) AND #pHsMx_3)) AND #pHsMx_4)) AND #EstadoZona.Marcha_CBx,   // "FB910_CNT_UHS"
                   R := (NOT #Mx_ET10 AND NOT #Mx_ET11 AND NOT #Mx_ET30 AND NOT #Mx_ET31) OR #TOut_Interlock.QU,
                   PV := #V_TOut_Interlock,
                   BaseUnidades_ms := "CTE_BaseUnidades_1s");
END_REGION

REGION Network 146: ERROR - Interlock con el FSS
   RUNG wire#powerrail
      Contact( #EstadoZona.Rearme_CBx )
      S_RS(operand := #EstadoVI.Err_Interlock_Salida, s1 := #TOut_Interlock.QU)
      S_Coil( #EstadoVI.Error_Mx )
   END_RUNG
   // the same network as SCL:
   IF #EstadoZona.Rearme_CBx THEN
       #EstadoVI.Err_Interlock_Salida := FALSE;   // RS flip-flop
   END_IF;
   IF #TOut_Interlock.QU THEN #EstadoVI.Err_Interlock_Salida := TRUE; END_IF;
   IF #EstadoVI.Err_Interlock_Salida THEN #EstadoVI.Error_Mx := TRUE; END_IF;
END_REGION

REGION Network 147: ESTADOS DE LA MESA
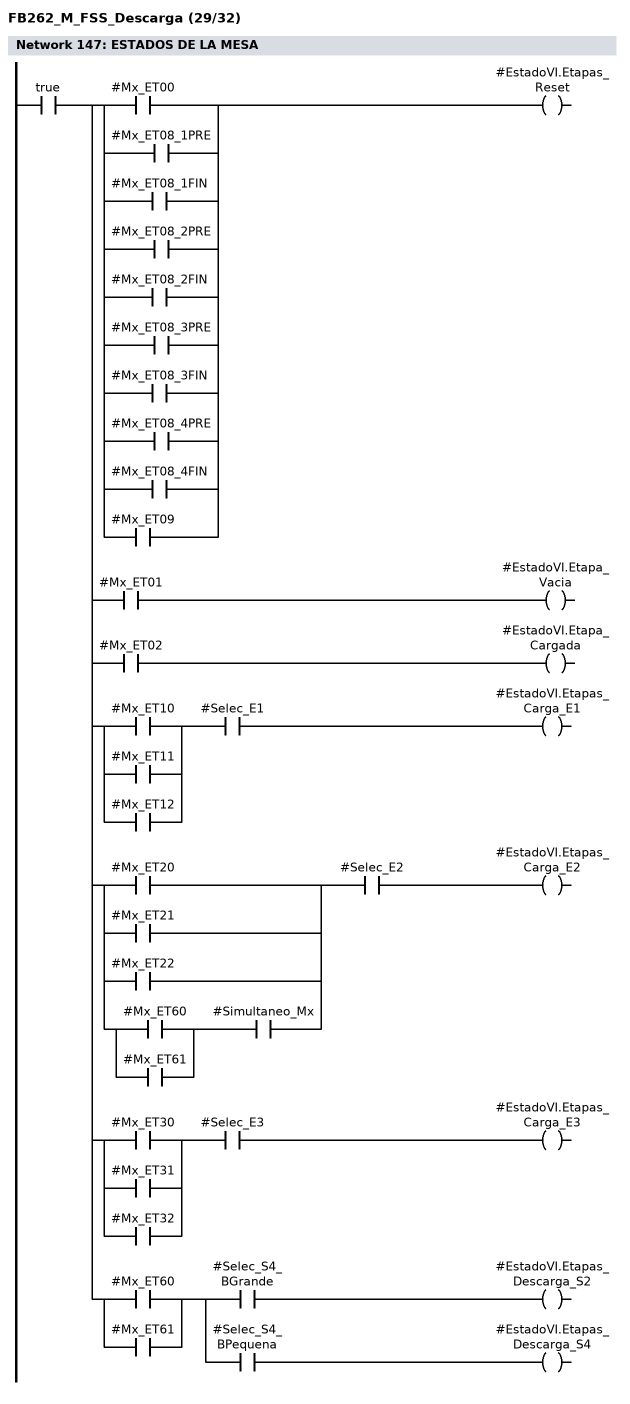
   RUNG wire#powerrail
      Contact( true )
      wire#w1
      Contact( #Mx_ET00 )
      wire#w2
      Coil( #EstadoVI.Etapas_Reset )
   END_RUNG
   RUNG wire#w1
      Contact( #Mx_ET08_1PRE )
   END_RUNG wire#w2
   RUNG wire#w1
      Contact( #Mx_ET08_1FIN )
   END_RUNG wire#w2
   RUNG wire#w1
      Contact( #Mx_ET08_2PRE )
   END_RUNG wire#w2
   RUNG wire#w1
      Contact( #Mx_ET08_2FIN )
   END_RUNG wire#w2
   RUNG wire#w1
      Contact( #Mx_ET08_3PRE )
   END_RUNG wire#w2
   RUNG wire#w1
      Contact( #Mx_ET08_3FIN )
   END_RUNG wire#w2
   RUNG wire#w1
      Contact( #Mx_ET08_4PRE )
   END_RUNG wire#w2
   RUNG wire#w1
      Contact( #Mx_ET08_4FIN )
   END_RUNG wire#w2
   RUNG wire#w1
      Contact( #Mx_ET09 )
   END_RUNG wire#w2
   RUNG wire#w1
      Contact( #Mx_ET01 )
      Coil( #EstadoVI.Etapa_Vacia )
   END_RUNG
   RUNG wire#w1
      Contact( #Mx_ET02 )
      Coil( #EstadoVI.Etapa_Cargada )
   END_RUNG
   RUNG wire#w1
      Contact( #Mx_ET10 )
      wire#w3
      Contact( #Selec_E1 )
      Coil( #EstadoVI.Etapas_Carga_E1 )
   END_RUNG
   RUNG wire#w1
      Contact( #Mx_ET11 )
   END_RUNG wire#w3
   RUNG wire#w1
      Contact( #Mx_ET12 )
   END_RUNG wire#w3
   RUNG wire#w1
      Contact( #Mx_ET20 )
      wire#w4
      Contact( #Selec_E2 )
      Coil( #EstadoVI.Etapas_Carga_E2 )
   END_RUNG
   RUNG wire#w1
      Contact( #Mx_ET21 )
   END_RUNG wire#w4
   RUNG wire#w1
      Contact( #Mx_ET22 )
   END_RUNG wire#w4
   RUNG wire#w1
      Contact( #Mx_ET60 )
      wire#w5
      Contact( #Simultaneo_Mx )
   END_RUNG wire#w4
   RUNG wire#w1
      Contact( #Mx_ET61 )
   END_RUNG wire#w5
   RUNG wire#w1
      Contact( #Mx_ET30 )
      wire#w6
      Contact( #Selec_E3 )
      Coil( #EstadoVI.Etapas_Carga_E3 )
   END_RUNG
   RUNG wire#w1
      Contact( #Mx_ET31 )
   END_RUNG wire#w6
   RUNG wire#w1
      Contact( #Mx_ET32 )
   END_RUNG wire#w6
   RUNG wire#w1
      Contact( #Mx_ET60 )
      wire#w7
      Contact( #Selec_S4_BGrande )
      Coil( #EstadoVI.Etapas_Descarga_S2 )
   END_RUNG
   RUNG wire#w1
      Contact( #Mx_ET61 )
   END_RUNG wire#w7
   RUNG wire#w7
      Contact( #Selec_S4_BPequena )
      Coil( #EstadoVI.Etapas_Descarga_S4 )
   END_RUNG
   // the same network as SCL:
   #EstadoVI.Etapas_Reset := true AND (#Mx_ET00 OR #Mx_ET08_1PRE OR #Mx_ET08_1FIN OR #Mx_ET08_2PRE OR #Mx_ET08_2FIN OR #Mx_ET08_3PRE OR #Mx_ET08_3FIN OR #Mx_ET08_4PRE OR #Mx_ET08_4FIN OR #Mx_ET09);
   #EstadoVI.Etapa_Vacia := true AND #Mx_ET01;
   #EstadoVI.Etapa_Cargada := true AND #Mx_ET02;
   #EstadoVI.Etapas_Carga_E1 := true AND (#Mx_ET10 OR #Mx_ET11 OR #Mx_ET12) AND #Selec_E1;
   #EstadoVI.Etapas_Carga_E2 := true AND (#Mx_ET20 OR #Mx_ET21 OR #Mx_ET22 OR ((#Mx_ET60 OR #Mx_ET61) AND #Simultaneo_Mx)) AND #Selec_E2;
   #EstadoVI.Etapas_Carga_E3 := true AND (#Mx_ET30 OR #Mx_ET31 OR #Mx_ET32) AND #Selec_E3;
   #_w1 := true AND (#Mx_ET60 OR #Mx_ET61);
   #EstadoVI.Etapas_Descarga_S2 := #_w1 AND #Selec_S4_BGrande;
   #EstadoVI.Etapas_Descarga_S4 := #_w1 AND #Selec_S4_BPequena;
END_REGION

REGION Network 148: ENTRADAS DE LA MESA
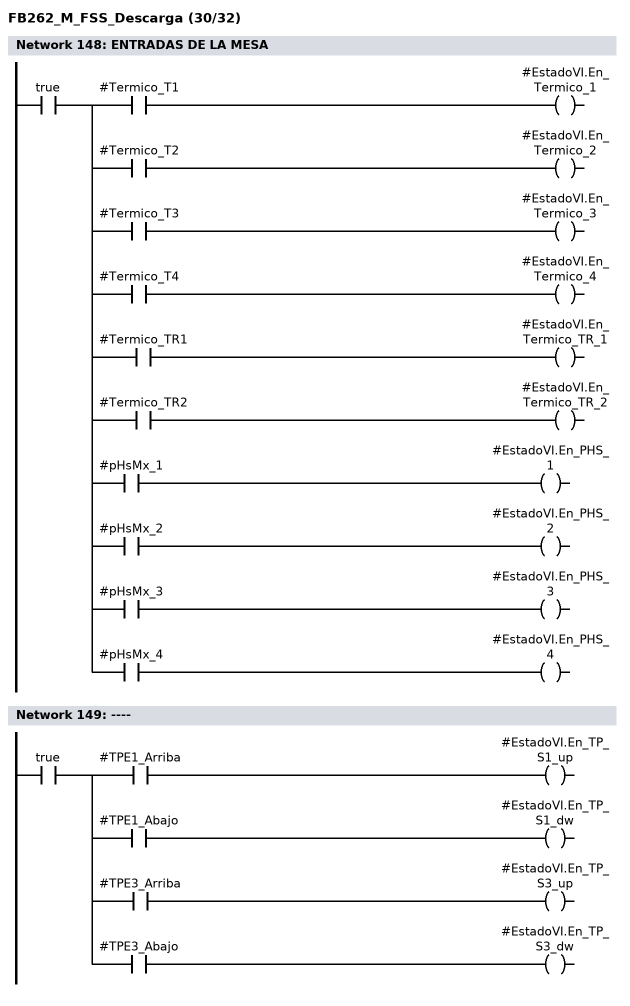
   RUNG wire#powerrail
      Contact( true )
      wire#w1
      Contact( #Termico_T1 )
      Coil( #EstadoVI.En_Termico_1 )
   END_RUNG
   RUNG wire#w1
      Contact( #Termico_T2 )
      Coil( #EstadoVI.En_Termico_2 )
   END_RUNG
   RUNG wire#w1
      Contact( #Termico_T3 )
      Coil( #EstadoVI.En_Termico_3 )
   END_RUNG
   RUNG wire#w1
      Contact( #Termico_T4 )
      Coil( #EstadoVI.En_Termico_4 )
   END_RUNG
   RUNG wire#w1
      Contact( #Termico_TR1 )
      Coil( #EstadoVI.En_Termico_TR_1 )
   END_RUNG
   RUNG wire#w1
      Contact( #Termico_TR2 )
      Coil( #EstadoVI.En_Termico_TR_2 )
   END_RUNG
   RUNG wire#w1
      Contact( #pHsMx_1 )
      Coil( #EstadoVI.En_PHS_1 )
   END_RUNG
   RUNG wire#w1
      Contact( #pHsMx_2 )
      Coil( #EstadoVI.En_PHS_2 )
   END_RUNG
   RUNG wire#w1
      Contact( #pHsMx_3 )
      Coil( #EstadoVI.En_PHS_3 )
   END_RUNG
   RUNG wire#w1
      Contact( #pHsMx_4 )
      Coil( #EstadoVI.En_PHS_4 )
   END_RUNG
   // the same network as SCL:
   #EstadoVI.En_Termico_1 := true AND #Termico_T1;
   #EstadoVI.En_Termico_2 := true AND #Termico_T2;
   #EstadoVI.En_Termico_3 := true AND #Termico_T3;
   #EstadoVI.En_Termico_4 := true AND #Termico_T4;
   #EstadoVI.En_Termico_TR_1 := true AND #Termico_TR1;
   #EstadoVI.En_Termico_TR_2 := true AND #Termico_TR2;
   #EstadoVI.En_PHS_1 := true AND #pHsMx_1;
   #EstadoVI.En_PHS_2 := true AND #pHsMx_2;
   #EstadoVI.En_PHS_3 := true AND #pHsMx_3;
   #EstadoVI.En_PHS_4 := true AND #pHsMx_4;
END_REGION

REGION Network 149: ----
   RUNG wire#powerrail
      Contact( true )
      wire#w1
      Contact( #TPE1_Arriba )
      Coil( #EstadoVI.En_TP_S1_up )
   END_RUNG
   RUNG wire#w1
      Contact( #TPE1_Abajo )
      Coil( #EstadoVI.En_TP_S1_dw )
   END_RUNG
   RUNG wire#w1
      Contact( #TPE3_Arriba )
      Coil( #EstadoVI.En_TP_S3_up )
   END_RUNG
   RUNG wire#w1
      Contact( #TPE3_Abajo )
      Coil( #EstadoVI.En_TP_S3_dw )
   END_RUNG
   // the same network as SCL:
   #EstadoVI.En_TP_S1_up := true AND #TPE1_Arriba;
   #EstadoVI.En_TP_S1_dw := true AND #TPE1_Abajo;
   #EstadoVI.En_TP_S3_up := true AND #TPE3_Arriba;
   #EstadoVI.En_TP_S3_dw := true AND #TPE3_Abajo;
END_REGION

REGION Network 150: SALIDAS de la Mesa
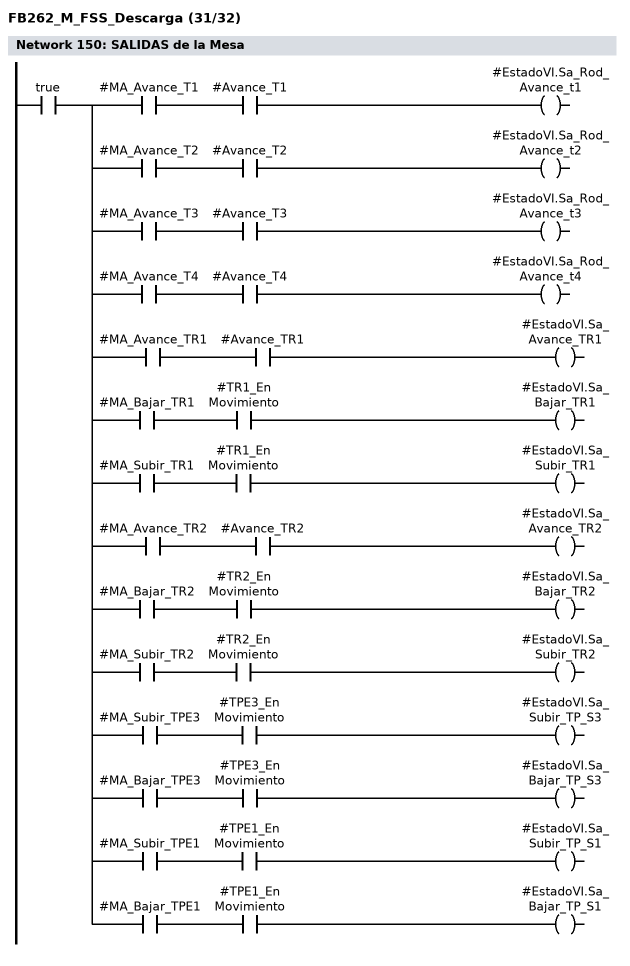
   RUNG wire#powerrail
      Contact( true )
      wire#w1
      Contact( #MA_Avance_T1 )
      Contact( #Avance_T1 )
      Coil( #EstadoVI.Sa_Rod_Avance_t1 )
   END_RUNG
   RUNG wire#w1
      Contact( #MA_Avance_T2 )
      Contact( #Avance_T2 )
      Coil( #EstadoVI.Sa_Rod_Avance_t2 )
   END_RUNG
   RUNG wire#w1
      Contact( #MA_Avance_T3 )
      Contact( #Avance_T3 )
      Coil( #EstadoVI.Sa_Rod_Avance_t3 )
   END_RUNG
   RUNG wire#w1
      Contact( #MA_Avance_T4 )
      Contact( #Avance_T4 )
      Coil( #EstadoVI.Sa_Rod_Avance_t4 )
   END_RUNG
   RUNG wire#w1
      Contact( #MA_Avance_TR1 )
      Contact( #Avance_TR1 )
      Coil( #EstadoVI.Sa_Avance_TR1 )
   END_RUNG
   RUNG wire#w1
      Contact( #MA_Bajar_TR1 )
      Contact( #TR1_EnMovimiento )
      Coil( #EstadoVI.Sa_Bajar_TR1 )
   END_RUNG
   RUNG wire#w1
      Contact( #MA_Subir_TR1 )
      Contact( #TR1_EnMovimiento )
      Coil( #EstadoVI.Sa_Subir_TR1 )
   END_RUNG
   RUNG wire#w1
      Contact( #MA_Avance_TR2 )
      Contact( #Avance_TR2 )
      Coil( #EstadoVI.Sa_Avance_TR2 )
   END_RUNG
   RUNG wire#w1
      Contact( #MA_Bajar_TR2 )
      Contact( #TR2_EnMovimiento )
      Coil( #EstadoVI.Sa_Bajar_TR2 )
   END_RUNG
   RUNG wire#w1
      Contact( #MA_Subir_TR2 )
      Contact( #TR2_EnMovimiento )
      Coil( #EstadoVI.Sa_Subir_TR2 )
   END_RUNG
   RUNG wire#w1
      Contact( #MA_Subir_TPE3 )
      Contact( #TPE3_EnMovimiento )
      Coil( #EstadoVI.Sa_Subir_TP_S3 )
   END_RUNG
   RUNG wire#w1
      Contact( #MA_Bajar_TPE3 )
      Contact( #TPE3_EnMovimiento )
      Coil( #EstadoVI.Sa_Bajar_TP_S3 )
   END_RUNG
   RUNG wire#w1
      Contact( #MA_Subir_TPE1 )
      Contact( #TPE1_EnMovimiento )
      Coil( #EstadoVI.Sa_Subir_TP_S1 )
   END_RUNG
   RUNG wire#w1
      Contact( #MA_Bajar_TPE1 )
      Contact( #TPE1_EnMovimiento )
      Coil( #EstadoVI.Sa_Bajar_TP_S1 )
   END_RUNG
   // the same network as SCL:
   #EstadoVI.Sa_Rod_Avance_t1 := true AND #MA_Avance_T1 AND #Avance_T1;
   #EstadoVI.Sa_Rod_Avance_t2 := true AND #MA_Avance_T2 AND #Avance_T2;
   #EstadoVI.Sa_Rod_Avance_t3 := true AND #MA_Avance_T3 AND #Avance_T3;
   #EstadoVI.Sa_Rod_Avance_t4 := true AND #MA_Avance_T4 AND #Avance_T4;
   #EstadoVI.Sa_Avance_TR1 := true AND #MA_Avance_TR1 AND #Avance_TR1;
   #EstadoVI.Sa_Bajar_TR1 := true AND #MA_Bajar_TR1 AND #TR1_EnMovimiento;
   #EstadoVI.Sa_Subir_TR1 := true AND #MA_Subir_TR1 AND #TR1_EnMovimiento;
   #EstadoVI.Sa_Avance_TR2 := true AND #MA_Avance_TR2 AND #Avance_TR2;
   #EstadoVI.Sa_Bajar_TR2 := true AND #MA_Bajar_TR2 AND #TR2_EnMovimiento;
   #EstadoVI.Sa_Subir_TR2 := true AND #MA_Subir_TR2 AND #TR2_EnMovimiento;
   #EstadoVI.Sa_Subir_TP_S3 := true AND #MA_Subir_TPE3 AND #TPE3_EnMovimiento;
   #EstadoVI.Sa_Bajar_TP_S3 := true AND #MA_Bajar_TPE3 AND #TPE3_EnMovimiento;
   #EstadoVI.Sa_Subir_TP_S1 := true AND #MA_Subir_TPE1 AND #TPE1_EnMovimiento;
   #EstadoVI.Sa_Bajar_TP_S1 := true AND #MA_Bajar_TPE1 AND #TPE1_EnMovimiento;
END_REGION

REGION Network 151: INTERLOCK PARA HMI
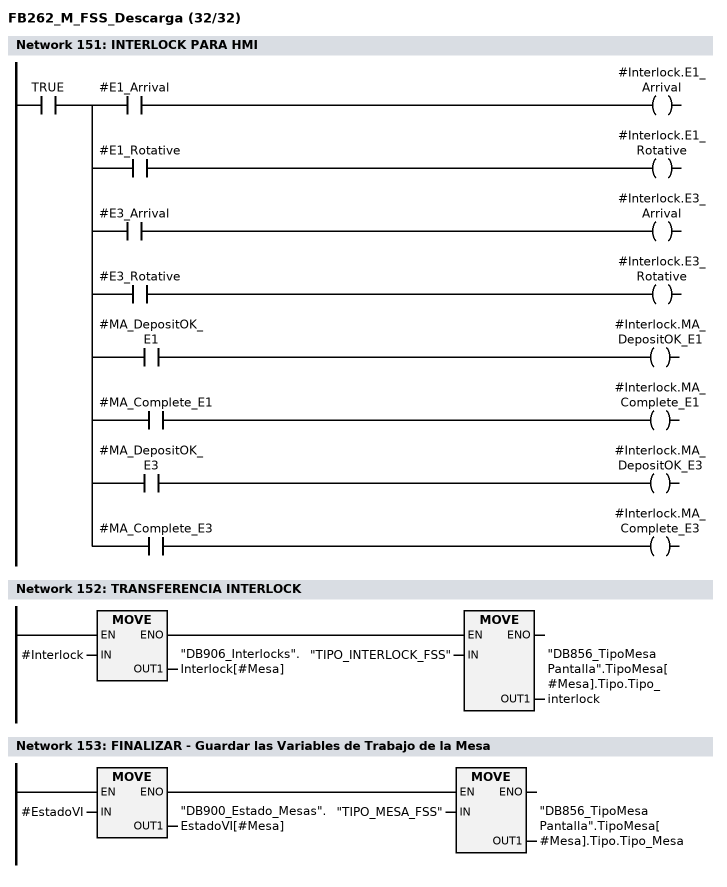
   RUNG wire#powerrail
      Contact( TRUE )
      wire#w1
      Contact( #E1_Arrival )
      Coil( #Interlock.E1_Arrival )
   END_RUNG
   RUNG wire#w1
      Contact( #E1_Rotative )
      Coil( #Interlock.E1_Rotative )
   END_RUNG
   RUNG wire#w1
      Contact( #E3_Arrival )
      Coil( #Interlock.E3_Arrival )
   END_RUNG
   RUNG wire#w1
      Contact( #E3_Rotative )
      Coil( #Interlock.E3_Rotative )
   END_RUNG
   RUNG wire#w1
      Contact( #MA_DepositOK_E1 )
      Coil( #Interlock.MA_DepositOK_E1 )
   END_RUNG
   RUNG wire#w1
      Contact( #MA_Complete_E1 )
      Coil( #Interlock.MA_Complete_E1 )
   END_RUNG
   RUNG wire#w1
      Contact( #MA_DepositOK_E3 )
      Coil( #Interlock.MA_DepositOK_E3 )
   END_RUNG
   RUNG wire#w1
      Contact( #MA_Complete_E3 )
      Coil( #Interlock.MA_Complete_E3 )
   END_RUNG
   // the same network as SCL:
   #Interlock.E1_Arrival := TRUE AND #E1_Arrival;
   #Interlock.E1_Rotative := TRUE AND #E1_Rotative;
   #Interlock.E3_Arrival := TRUE AND #E3_Arrival;
   #Interlock.E3_Rotative := TRUE AND #E3_Rotative;
   #Interlock.MA_DepositOK_E1 := TRUE AND #MA_DepositOK_E1;
   #Interlock.MA_Complete_E1 := TRUE AND #MA_Complete_E1;
   #Interlock.MA_DepositOK_E3 := TRUE AND #MA_DepositOK_E3;
   #Interlock.MA_Complete_E3 := TRUE AND #MA_Complete_E3;
END_REGION

REGION Network 152: TRANSFERENCIA INTERLOCK
   RUNG wire#powerrail
      Move(in := #Interlock, out1 => "DB906_Interlocks".Interlock[#Mesa])
      Move(in := "TIPO_INTERLOCK_FSS", out1 => "DB856_TipoMesaPantalla".TipoMesa[#Mesa].Tipo.Tipo_interlock)
   END_RUNG
   // the same network as SCL:
   "DB906_Interlocks".Interlock[#Mesa] := #Interlock;
   "DB856_TipoMesaPantalla".TipoMesa[#Mesa].Tipo.Tipo_interlock := "TIPO_INTERLOCK_FSS";
END_REGION

REGION Network 153: FINALIZAR - Guardar las Variables de Trabajo de la Mesa
   RUNG wire#powerrail
      Move(in := #EstadoVI, out1 => "DB900_Estado_Mesas".EstadoVI[#Mesa])
      Move(in := "TIPO_MESA_FSS", out1 => "DB856_TipoMesaPantalla".TipoMesa[#Mesa].Tipo.Tipo_Mesa)
   END_RUNG
   // the same network as SCL:
   "DB900_Estado_Mesas".EstadoVI[#Mesa] := #EstadoVI;
   "DB856_TipoMesaPantalla".TipoMesa[#Mesa].Tipo.Tipo_Mesa := "TIPO_MESA_FSS";
END_REGION
END_FUNCTION_BLOCK
